(* PLC project Generated.project, CODESYS CODESYS V3.5 SP19 Patch 1 *)
(* stored: creationDateTime 2026-08-11T18:19:14.795164, modificationDateTime 2026-08-11T18:19:14.795164 *)

(* ═══════════════════════════════════════════════════════════════════════════════ 📊 ST_WinchLoadEstimateTable — Table empirique charge estimée ═══════════════════════════════════════════════════════════════════════════════ ⚠️ Valeur informative uniquement : ce tableau ne remplace pas une mesure de charge certifiée et ne participe à aucune fonction de sécurité. 🧭 Index 1 : palier contacteurs commandé (1..5) 🧭 Index 2 : bande de vitesse câble mesurée (1..5) 📐 Valeur : estimation charge en pourcentage (0..100 %), réglée sur site. ═══════════════════════════════════════════════════════════════════════════════ 📄 Docs : DOC/AF/AF_Partie-10_Fonction_Winch_v2.0.md *)
TYPE ST_WinchLoadEstimateTable : STRUCT
  IsConfigured : BOOL;
  LoadPctByStepAndSpeedBand : ARRAY[1..5] OF ARRAY[1..5] OF REAL;  (* 🔧 Tableau imbriqué (accès [palier][bande]) — le multi-dim ARRAY[x,y] n'est pas supporté par TOOLS/ST_PLCOPENXML_GENERATOR *)
END_STRUCT;
END_TYPE
